INTERFACE ITF_pompdigout

METHOD set : bool
VAR_INPUT
	state : BOOL;
END_VAR
END_METHOD

END_INTERFACE

(* stored: Version 1.1.0.1, ProductVersion 3.1.4026.8
   Itf ITF_pompdigout: Id {11ce1814-e1e2-4478-bbb0-4699c4add5ba}
   Method set: Id {6a1cfa76-3656-4d97-ae72-2b3d1fac0981} *)
